{attribute 'linkalways'} 
{attribute 'no_explicit_call' := 'This FB is a CLASS and must be accessed using methods or properties'}
{attribute 'enable_dynamic_creation'}
FUNCTION_BLOCK Node_ContainerType_Vector_Vector_TcVnPoint3_REAL EXTENDS Node
VAR
    out : _GUID;
END_VAR

METHOD PUBLIC  Clone : I_Node
VAR
	pNode : POINTER TO Node_ContainerType_Vector_Vector_TcVnPoint3_REAL;
END_VAR
pNode := __NEW(Node_ContainerType_Vector_Vector_TcVnPoint3_REAL);
Clone := pNode^;
END_METHOD

METHOD FB_init : BOOL
VAR_INPUT
	bInitRetains : BOOL; // if TRUE, the retain variables are initialized (warm start / cold start)
	bInCopyCode : BOOL;  // if TRUE, the instance afterwards gets moved into the copy code (online change)
END_VAR
AddOutput('out', out);
END_METHOD

METHOD PROTECTED OnExecute
out.Value := ContainerType_Vector_Vector_TcVnPoint3_REAL;
END_METHOD

END_FUNCTION_BLOCK

(* stored: Version 1.1.0.1, ProductVersion 3.1.4026.17
   POU Node_ContainerType_Vector_Vector_TcVnPoint3_REAL: Id {1d908790-3d2f-02b7-300a-e047d5a4d0d8}, SpecialFunc None
   Folder Constructor: Id {d4d2a272-e5e5-0d1a-0cbf-58d050e57c83}
   Method Clone: Id {823a58fb-5bd3-0b37-3b47-fcf19321cfbe}
   Method FB_init: Id {a25c5275-393e-001e-06e7-ea88da7ea155}
   Method OnExecute: Id {614e180f-e268-043a-092c-11a225c7c5b6} *)
